PROGRAM Decoder
VAR
END_VAR

END_PROGRAM

(* stored: Version 1.1.0.1, ProductVersion 3.1.4024.0
   POU Decoder: Id {1cfc5b98-9cc8-438c-ae60-709acd6a425e}, SpecialFunc None *)
